{attribute 'qualified_only'}
{attribute 'strict'}
{attribute 'to_string'}

TYPE E_RequestState :
(
	{attribute 'hide'}
    Undefined   := 0,
	{attribute 'analysis' := '-27'}
	Reset       := 1,
	{attribute 'analysis' := '-27'}
    Start       := 2,
    Hold      	:= 4,
	Stop		:= 8,
	Abort       := 16
);
END_TYPE

(* stored: Version 1.1.0.1
   DUT E_RequestState: Id {d3b20770-b5da-468b-8276-148bae048ad0} *)
